PROGRAM EXAMPLES_PRG
VAR
	_context : fbContext;
	_recordableStations : RecordableStation001;
	_loggerContext : LoggerContext;
	_strucuredContext : StrucuredContext;
	a : TcoCore.ITcoObject;
END_VAR

_context.Run();
_recordableStations.Run();
_loggerContext.Run();

a := _strucuredContext._structuredData._o1.Parent;

END_PROGRAM

(* stored: Version 1.1.0.1
   POU EXAMPLES_PRG: Id {ce53afe8-e524-0dc9-2ef6-f4e12a5dd130}, SpecialFunc None *)
